// TIA Portal V17 export
// export: Created 2023-02-23T17:16:27.747253Z, ExportSetting WithDefaults, DisplayName Totally Integrated Automation Portal, DisplayVersion V17, DisplayName TIA Portal Openness, DisplayVersion V17, DisplayName TIA Portal Version Control Interface, DisplayVersion V17, DisplayName TIA Portal Test Suite Advanced, DisplayVersion V17, DisplayName STEP 7 Professional, DisplayVersion V17, DisplayName SIMATIC Energy Suite, DisplayVersion V17, DisplayName STEP 7 Safety, DisplayVersion V17, DisplayName WinCC Professional, DisplayVersion V17
FUNCTION "TST_ClassTest" : Void   // FC2, LAD
{ S7_Optimized_Access := 'TRUE' }
VERSION : 0.1
// stored: AutoNumber true, IsIECCheckEnabled false, SetENOAutomatically false, UDAEnableTagReadback false
BEGIN

REGION Network 1: Call: ChooseMode
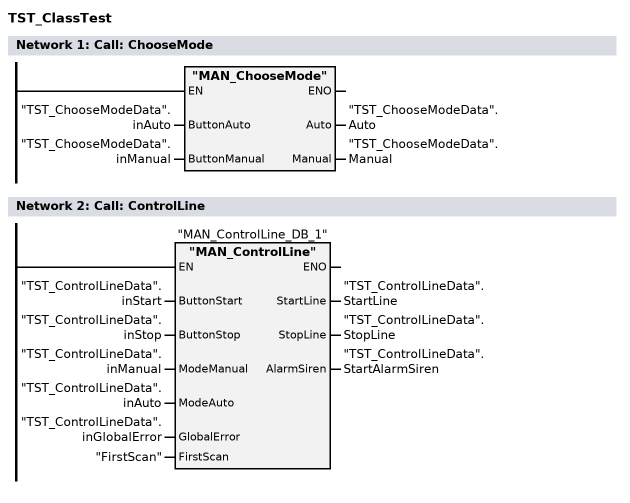
   RUNG wire#powerrail
      "MAN_ChooseMode"(ButtonAuto := "TST_ChooseModeData".inAuto, ButtonManual := "TST_ChooseModeData".inManual, Auto => "TST_ChooseModeData".Auto, Manual => "TST_ChooseModeData".Manual)
   END_RUNG
   // the same network as SCL:
   "MAN_ChooseMode"(ButtonAuto := "TST_ChooseModeData".inAuto,
                    ButtonManual := "TST_ChooseModeData".inManual,
                    Auto => "TST_ChooseModeData".Auto,
                    Manual => "TST_ChooseModeData".Manual);
END_REGION

REGION Network 2: Call: ControlLine
   RUNG wire#powerrail
      "MAN_ControlLine_DB_1"(ButtonStart := "TST_ControlLineData".inStart, ButtonStop := "TST_ControlLineData".inStop, ModeManual := "TST_ControlLineData".inManual, ModeAuto := "TST_ControlLineData".inAuto, GlobalError := "TST_ControlLineData".inGlobalError, FirstScan := "FirstScan", StartLine => "TST_ControlLineData".StartLine, StopLine => "TST_ControlLineData".StopLine, AlarmSiren => "TST_ControlLineData".StartAlarmSiren)
   END_RUNG
   // the same network as SCL:
   "MAN_ControlLine_DB_1"(ButtonStart := "TST_ControlLineData".inStart,   // "MAN_ControlLine"
                          ButtonStop := "TST_ControlLineData".inStop,
                          ModeManual := "TST_ControlLineData".inManual,
                          ModeAuto := "TST_ControlLineData".inAuto,
                          GlobalError := "TST_ControlLineData".inGlobalError,
                          FirstScan := "FirstScan",
                          StartLine => "TST_ControlLineData".StartLine,
                          StopLine => "TST_ControlLineData".StopLine,
                          AlarmSiren => "TST_ControlLineData".StartAlarmSiren);
END_REGION
END_FUNCTION
